// Comparison enum.
{attribute 'qualified_only'}
{attribute 'to_string'}
TYPE E_Comparison :
(
	_ := 0, // Unknown/Invalid
	Less,
	Equal,
	Greater
)BYTE;
END_TYPE

(* stored: Version 1.1.0.1
   EnumerationTextList E_Comparison: Id {35f4561f-4e16-044f-02b6-7f4c15b97f0a} *)
